SUBAPPLICATION Uebung_039_sub_Outputs (* Subapplication Type *)
  (* Standard: 61499-2 *)
  (* Version 1.0, 2024-03-03, franz *)
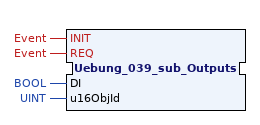
  EVENT_INPUT
    INIT; (* Service Initialization *)
    REQ; (* Service Request *)
  END_EVENT
  VAR_INPUT
    DI : BOOL; (* Digital Input *)
    u16ObjId : UINT := ID_NULL; (* Object ID Softkey/Button *)
  END_VAR
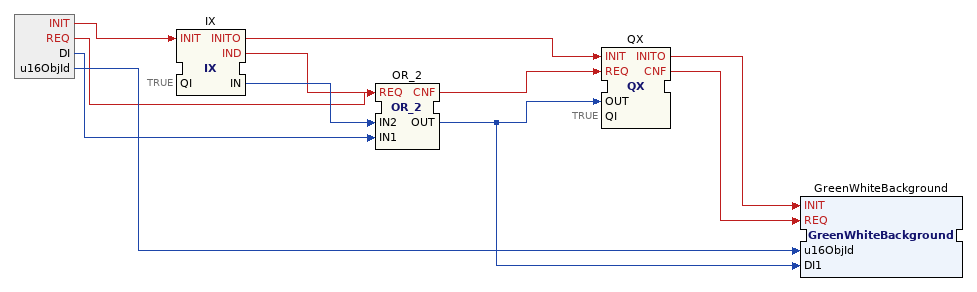
  FBS
    QX : QX(QI := TRUE);
    IX : IX(QI := TRUE);
    OR_2 : OR_2;
  END_FBS
  SUBAPPS
    GreenWhiteBackground : GreenWhiteBackground;
  END_SUBAPPS
  EVENT_CONNECTIONS
    IX.INITO TO QX.INIT;
    INIT TO IX.INIT;
    QX.INITO TO GreenWhiteBackground.INIT;
    QX.CNF TO GreenWhiteBackground.REQ;
    OR_2.CNF TO QX.REQ;
    IX.IND TO OR_2.REQ;
    REQ TO OR_2.REQ;
  END_CONNECTIONS
  DATA_CONNECTIONS
    u16ObjId TO GreenWhiteBackground.u16ObjId;
    OR_2.OUT TO GreenWhiteBackground.DI1;
    OR_2.OUT TO QX.OUT;
    IX.IN TO OR_2.IN2;
    DI TO OR_2.IN1;
  END_CONNECTIONS
END_SUBAPPLICATION
